FUNCTION_BLOCK Throttle
  (* Standard: 61499-2 *)
  (* Version 0.2, 2003-12-04, JHC, Rockwell Automation, Renamed for better indexing. *)
  (* Version 0.1, 2002-11-05, JHC, Rockwell Automation, Corrected missing ST element in Algorithm REQ. *)
  (* Version 0.0, 2000-05-30, JHC, Rockwell Automation *)
  (* Compiler header: package fb.rt.benchmarks.cruisecontrol; *)
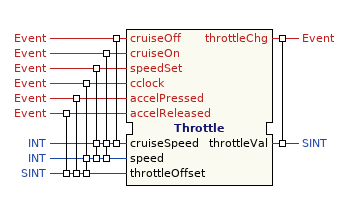
  EVENT_INPUT
    cruiseOff WITH cruiseSpeed;
    cruiseOn WITH cruiseSpeed, speed;
    speedSet WITH cruiseSpeed, speed;
    cclock WITH speed, throttleOffset; (* 10ms tick *)
    accelPressed WITH throttleOffset;
    accelReleased WITH throttleOffset;
  END_EVENT
  EVENT_OUTPUT
    throttleChg WITH throttleVal;
  END_EVENT
  VAR_INPUT
    cruiseSpeed : INT := 0; (* desired speed *)
    speed : INT := 0; (* actual speed *)
    throttleOffset : SINT := 0; (* offset angle *)
  END_VAR
  VAR_OUTPUT
    throttleVal : SINT := 0; (* throttle angle *)
  END_VAR
  VAR
    prevOffset : int := 0;
    tmp : int := 0;
  END_VAR
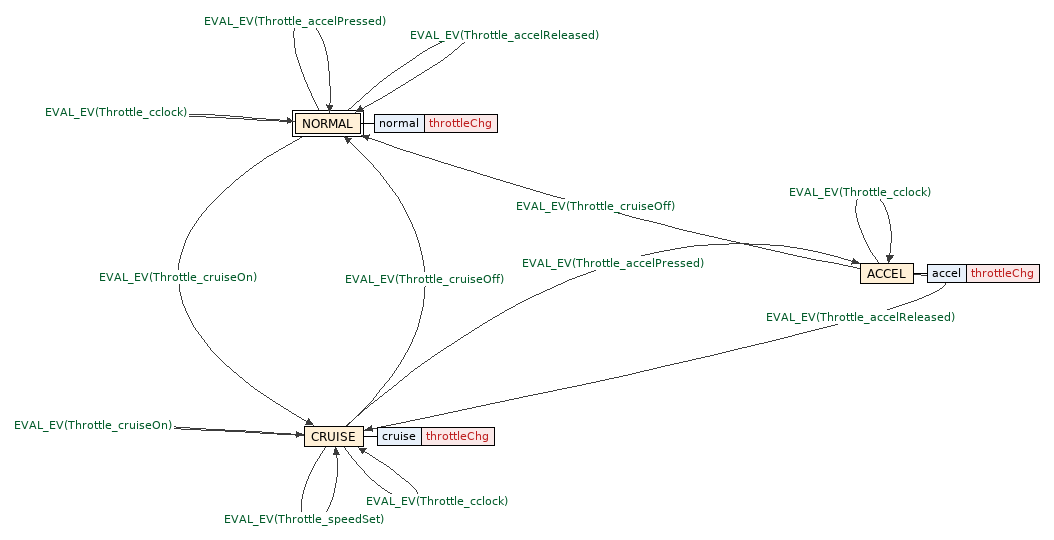
  EC_STATES
    NORMAL : normal -> throttleChg;
    CRUISE : cruise -> throttleChg;
    ACCEL : accel -> throttleChg;
  END_STATES
  EC_TRANSITIONS
    NORMAL TO CRUISE := EVAL_EV(Throttle_cruiseOn);
    NORMAL TO NORMAL := EVAL_EV(Throttle_accelPressed);
    NORMAL TO NORMAL := EVAL_EV(Throttle_accelReleased);
    NORMAL TO NORMAL := EVAL_EV(Throttle_cclock);
    CRUISE TO NORMAL := EVAL_EV(Throttle_cruiseOff);
    CRUISE TO ACCEL := EVAL_EV(Throttle_accelPressed);
    CRUISE TO CRUISE := EVAL_EV(Throttle_cruiseOn);
    CRUISE TO CRUISE := EVAL_EV(Throttle_speedSet);
    CRUISE TO CRUISE := EVAL_EV(Throttle_cclock);
    ACCEL TO NORMAL := EVAL_EV(Throttle_cruiseOff);
    ACCEL TO CRUISE := EVAL_EV(Throttle_accelReleased);
    ACCEL TO ACCEL := EVAL_EV(Throttle_cclock);
  END_TRANSITIONS
  ALGORITHM normal IN ST:
VAL_OF_throttleVal() = VAL_OF_throttleOffset();
prevOffset= 0;
  END_ALGORITHM
  ALGORITHM accel IN ST:
VAL_OF_throttleVal() = VAL_OF_throttleVal() + VAL_OF_throttleOffset() - prevOffset;
prevOffset= VAL_OF_throttleOffset();
  END_ALGORITHM
  ALGORITHM cruise IN ST:
tmp  = (VAL_OF_cruiseSpeed() - VAL_OF_speed());
tmp = tmp * 3;
 if (tmp > 45) {
    tmp = 45;
}else if( tmp < 0) {
    tmp = 0;
 };
 VAL_OF_throttleVal() = tmp;
  END_ALGORITHM
END_FUNCTION_BLOCK
